(* IEC 61131-3 sources: CodesysTest/alpha/export/Pro18_1174.dev/Plc Logic/Application/Motors/Applied Motion/FB_AppliedMotionBagDeliveryMotor_1.pou, 1 file *)

(* ---- MoveDistanceFinal.m.st ---- *)
(*#-#-#-#-#-#-#-#-#-#---Declaration---#-#-#-#-#-#-#-#-#-#-#-#-#*)

METHOD MoveDistanceFinal
VAR_INPUT
    distance : REAL;        //Distance to move in inches
    acceleration : INT;        //Acceleration in RPM/sec
    deceleration : INT;        //Deceleration in RPM/sec
    velocity : INT;            //Velocity in .25RPM
END_VAR
(*#-#-#-#-#-#-#-#-#-#---Implementation---#-#-#-#-#-#-#-#-#-#-#-#-#*)

commandSuccessful := FALSE;
_moveDone := FALSE;
moveDistanceFinalState := AMP_EIP_MOVE_INITIAL_STATES.Idle;
distanceToMoveInSteps := REAL_TO_DINT((distance) * stepsPerInchSetpoint);
IF reversePolarity THEN
    distanceToMoveInSteps := distanceToMoveInSteps * -1;
END_IF

pointToPointAccelSetpoint := acceleration;
pointToPointDecelSetpoint := deceleration;
velocitySetpoint := velocity;

currentLimit := defaultCurrentSetpoint;
_moveFinal := TRUE;
//SUPER^.ExecuteStoredProgram(2);
